// Mitsubishi GX Works2 project: 1   PLC: FX3U/FX3UC

// task Task_01 (event TRUE, interval 0, priority 31): POU_01

PROGRAM POU_01
VAR
  ton1 : TON;
END_VAR
ton1(IN := M0, PT := T#1s);
Y0 := ton1.Q;
END_PROGRAM
